FUNCTION "ST10_Alarm" : Void
VAR_TEMP
  tpAlarm : Array[0..2, 0..15] of Bool;
  tpAlarmInt : Array[0..2] of Int;
  tpTP : Array[0..1] of Int;
  tpClear : Byte;
  FixtureNumber : Int;
  i : Int;
  tpAlwayoff : Bool;
END_VAR
BEGIN
  // Původní jazyk: LAD
  // Zdroj XML: EXPORT/Program blocks/OP010/05_Alarm/ST10_Alarm.xml
  // (Žádný StructuredText network nebyl nalezen; LAD/STL/GRAPH není automaticky překládán.)
END_FUNCTION
